(* PLC project  *)

CONFIGURATION FSLOGIC
END_CONFIGURATION
